# EPICS IOC start-up script: iocsh/esschic.iocsh
#  ### esschic iocsh  ###
#- ###################################################
#-
#- CHIC_SYS       - Required: System prefix for CHIC PV names
#  CHIC_DEV	  - Required: Device name for CHIC PV names
#
#  TODO: Check CHOP_DRV definition
#- CHOP_DRV       - Required: Chopper drive PV name (device part)
#
#  TODO: Check SYS component
#- SYS            - Required: System prefix (for which component?)
#

dbLoadRecords("esschicTimestampBuffer.db", "CHIC_SYS=$(CHIC_SYS), CHOP_DRV=$(CHOP_DRV), SYS=$(SYS), DEVICE=$(CHIC_DEV):")
